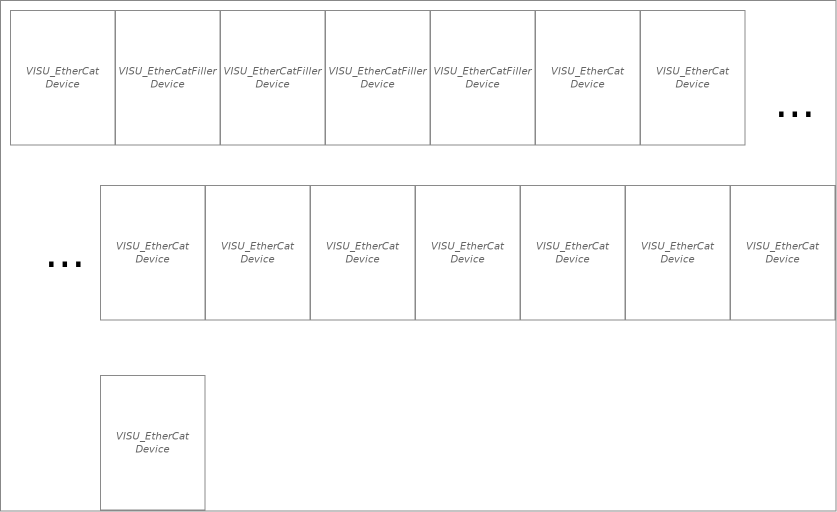
VISUALIZATION VISU_TelemetryIO  // 837x512
VAR_IN_OUT
	ref : TelemetryIO;
    widget : TelemetryIOWidget;
END_VAR
    Frame (10,10 105x135)
        shows VISU_EtherCatDevice(device := ref.parts.coupler, widget := widget.coupler)
    Frame (535,10 105x135)
        shows VISU_EtherCatDevice(device := ref.parts.slot5, widget := widget.slot5)
    Frame (520,185 105x135)
        shows VISU_EtherCatDevice(device := ref.parts.slot11, widget := widget.slot11)
    Frame (640,10 105x135)
        shows VISU_EtherCatDevice(device := ref.parts.slot6, widget := widget.slot6)
    Frame (625,185 105x135)
        shows VISU_EtherCatDevice(device := ref.parts.slot12, widget := widget.slot12)
    Frame (100,185 105x135)
        shows VISU_EtherCatDevice(device := ref.parts.slot7, widget := widget.slot7)
    Frame (730,185 105x135)
        shows VISU_EtherCatDevice(device := ref.parts.slot13, widget := widget.slot13)
    Frame (205,185 105x135)
        shows VISU_EtherCatDevice(device := ref.parts.slot8, widget := widget.slot8)
    Frame (310,185 105x135)
        shows VISU_EtherCatDevice(device := ref.parts.slot9, widget := widget.slot9)
    Frame (415,185 105x135)
        shows VISU_EtherCatDevice(device := ref.parts.slot10, widget := widget.slot10)
    Frame (115,10 105x135)
        shows VISU_EtherCatFillerDevice()
    Frame (220,10 105x135)
        shows VISU_EtherCatFillerDevice()
    Frame (325,10 105x135)
        shows VISU_EtherCatFillerDevice()
    Frame (430,10 105x135)
        shows VISU_EtherCatFillerDevice()
    Label (765,70 60x64), "..."
    Label (35,220 60x64), "..."
    Frame (100,375 105x135)
        shows VISU_EtherCatDevice(device := ref.parts.tubeAccelerometers, widget := widget.tubeAccelerometers)
END_VISUALIZATION

(* stored: Version 1.1.0.1, ProductVersion 3.1.4019.2
   Visu VISU_TelemetryIO: Id {cd2bba65-5a22-4a5c-8c0c-380800419611} *)
